{attribute 'GeneratedUsingTerminal: KL6301-0002'}
{attribute addProperty BoxType "KL6301-0002"}
{attribute addProperty Id "Channel_1AT %Q*Channel_9BC0092E0"}
{attribute addProperty CRC "942227994"}
{attribute addProperty Size "0"}
TYPE KL_3829421A :
STRUCT
	{attribute addProperty Name "Channel_1"}
	Channel_1 : Channel_9BC0092E;
END_STRUCT
END_TYPE

(* stored: Version 1.2.0.0, ProductVersion 3.1.4024.9
   DUT KL_3829421A: Id {c7556eeb-2c2f-4e02-8682-2f71d9d0a365} *)
